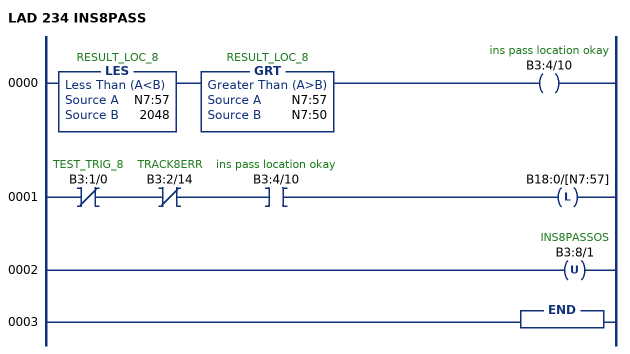
% Rung: 0 %
SOR LES N7:57 2048 GRT N7:57 N7:50 OTE B3:4/10 EOR
%   N7:57  RESULT_LOC_8 %
%   N7:50  INS_8_TRIG_LOC %
%   B3:4/10  "ins pass location okay" %
% Rung: 1 %
SOR XIO B3:1/0 XIO B3:2/14 XIC B3:4/10 OTL B18:0/[N7:57] EOR
%   B3:1/0  TEST_TRIG_8 %
%   B3:2/14  TRACK8ERR %
%   B3:4/10  "ins pass location okay" %
%   B18:0  GOOD2 %
%   N7:57  RESULT_LOC_8 %
% Rung: 2 %
SOR OTU B3:8/1 EOR
%   B3:8/1  INS8PASSOS %
% Rung: 3 %
SOR END EOR

LADDER 235 "INS8FAIL"
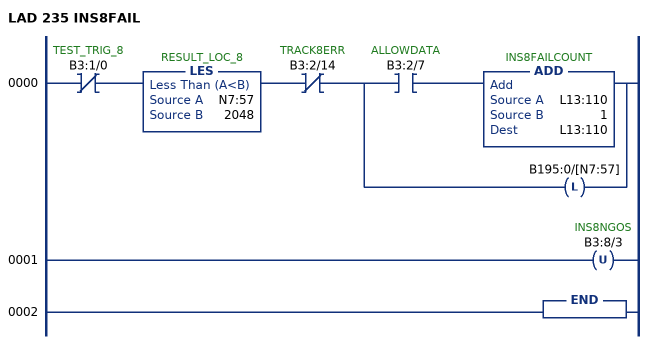
% Rung: 0 %
SOR XIO B3:1/0 LES N7:57 2048 XIO B3:2/14 BST XIC B3:2/7 ADD L13:110 1 L13:110 NXB OTL B195:0/[N7:57] BND EOR
%   B3:1/0  TEST_TRIG_8 %
%   N7:57  RESULT_LOC_8 %
%   B3:2/14  TRACK8ERR %
%   B3:2/7  ALLOWDATA %
%   L13:110  INS8FAILCOUNT %
%   B195:0  TOP_NG %
% Rung: 1 %
SOR OTU B3:8/3 EOR
%   B3:8/3  INS8NGOS %
% Rung: 2 %
SOR END EOR

LADDER 236 "INS8ACQ"
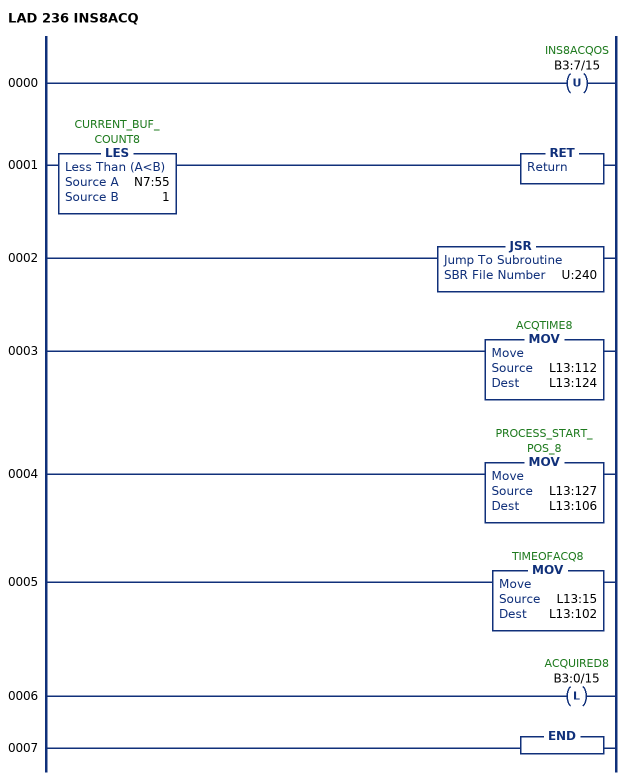
% Rung: 0 %
SOR OTU B3:7/15 EOR
%   B3:7/15  INS8ACQOS %
% Rung: 1 %
SOR LES N7:55 1 RET EOR
%   N7:55  CURRENT_BUF_COUNT8 %
% Rung: 2 %
SOR JSR U:240 EOR
% Rung: 3 %
SOR MOV L13:112 L13:124 EOR
%   L13:112  TIME_SPAN8 %
%   L13:124  ACQTIME8 %
% Rung: 4 %
SOR MOV L13:127 L13:106 EOR
%   L13:127  PULLED_POSITION8 %
%   L13:106  PROCESS_START_POS_8 %
% Rung: 5 %
SOR MOV L13:15 L13:102 EOR
%   L13:15  TOP_TIME %
%   L13:102  TIMEOFACQ8 %
% Rung: 6 %
SOR OTL B3:0/15 EOR
%   B3:0/15  ACQUIRED8 %
% Rung: 7 %
SOR END EOR

LADDER 237 "Q8TIMETEST"
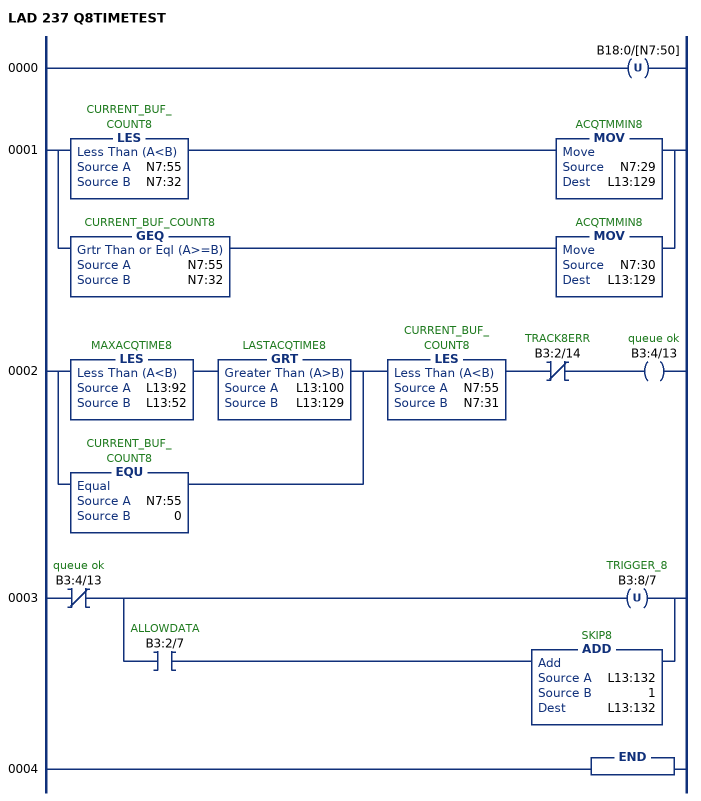
% Rung: 0 %
SOR OTU B18:0/[N7:50] EOR
%   B18:0  GOOD2 %
%   N7:50  INS_8_TRIG_LOC %
% Rung: 1 %
SOR BST LES N7:55 N7:32 MOV N7:29 L13:129 NXB GEQ N7:55 N7:32 MOV N7:30 L13:129 BND EOR
%   N7:55  CURRENT_BUF_COUNT8 %
%   N7:32  BUF_CAM_LIMIT %
%   N7:29  CAM_BUF_ACQ_TM %
%   L13:129  ACQTMMIN8 %
%   N7:30  PC_BUF_ACQ_TM %
% Rung: 2 %
SOR BST LES L13:92 L13:52 GRT L13:100 L13:129 NXB EQU N7:55 0 BND LES N7:55 N7:31 XIO B3:2/14 OTE B3:4/13 EOR
%   L13:92  MAXACQTIME8 %
%   L13:52  ACQTIMELIMIT %
%   L13:100  LASTACQTIME8 %
%   L13:129  ACQTMMIN8 %
%   N7:55  CURRENT_BUF_COUNT8 %
%   N7:31  MAX_BUFF_CT  "maximum buffers" %
%   B3:2/14  TRACK8ERR %
%   B3:4/13  "queue ok" %
% Rung: 3 %
SOR XIO B3:4/13 BST OTU B3:8/7 NXB XIC B3:2/7 ADD L13:132 1 L13:132 BND EOR
%   B3:4/13  "queue ok" %
%   B3:8/7  TRIGGER_8 %
%   B3:2/7  ALLOWDATA %
%   L13:132  SKIP8 %
% Rung: 4 %
SOR END EOR

LADDER 238 "INS8TRIG"
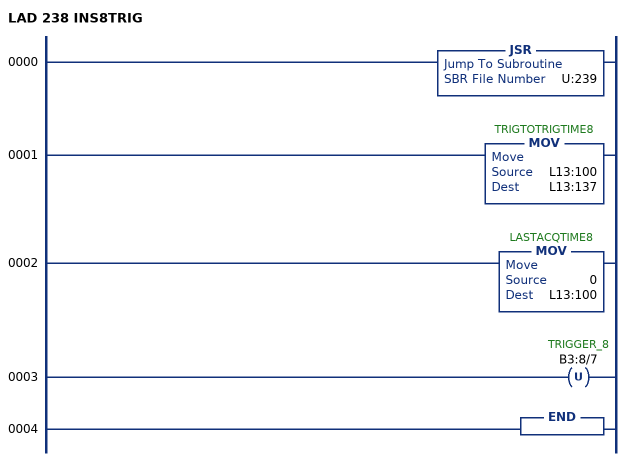
% Rung: 0 %
SOR JSR U:239 EOR
% Rung: 1 %
SOR MOV L13:100 L13:137 EOR
%   L13:100  LASTACQTIME8 %
%   L13:137  TRIGTOTRIGTIME8 %
% Rung: 2 %
SOR MOV 0 L13:100 EOR
%   L13:100  LASTACQTIME8 %
% Rung: 3 %
SOR OTU B3:8/7 EOR
%   B3:8/7  TRIGGER_8 %
% Rung: 4 %
SOR END EOR

LADDER 239 "FIFO8SET"
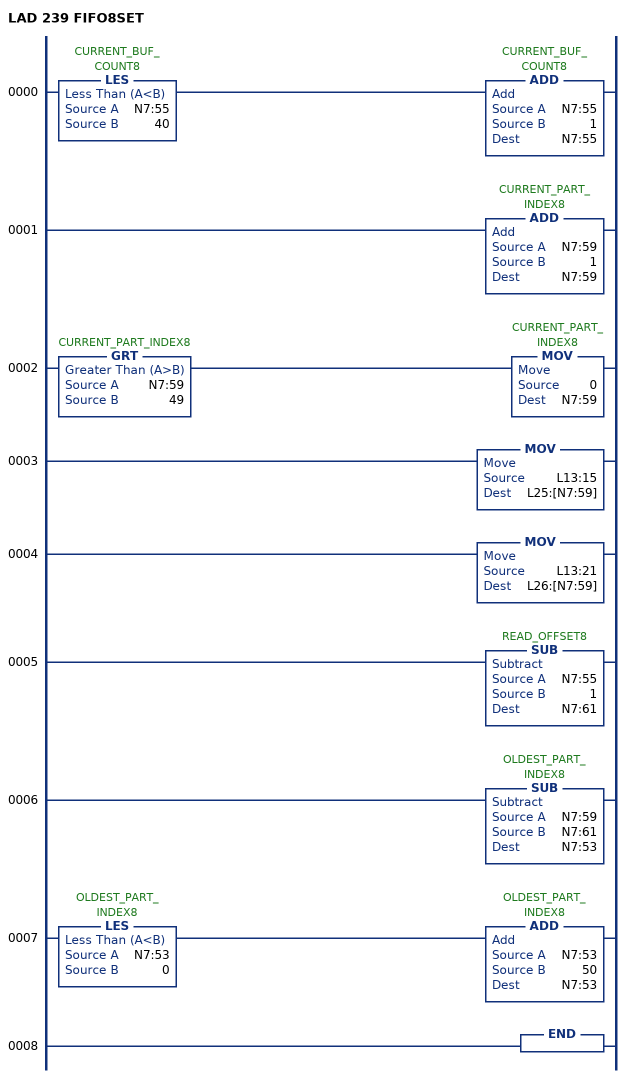
% Rung: 0 %
SOR LES N7:55 40 ADD N7:55 1 N7:55 EOR
%   N7:55  CURRENT_BUF_COUNT8 %
% Rung: 1 %
SOR ADD N7:59 1 N7:59 EOR
%   N7:59  CURRENT_PART_INDEX8 %
% Rung: 2 %
SOR GRT N7:59 49 MOV 0 N7:59 EOR
%   N7:59  CURRENT_PART_INDEX8 %
% Rung: 3 %
SOR MOV L13:15 L25:[N7:59] EOR
%   L13:15  TOP_TIME %
%   N7:59  CURRENT_PART_INDEX8 %
% Rung: 4 %
SOR MOV L13:21 L26:[N7:59] EOR
%   L13:21  TOP_POSITION %
%   N7:59  CURRENT_PART_INDEX8 %
% Rung: 5 %
SOR SUB N7:55 1 N7:61 EOR
%   N7:55  CURRENT_BUF_COUNT8 %
%   N7:61  READ_OFFSET8 %
% Rung: 6 %
SOR SUB N7:59 N7:61 N7:53 EOR
%   N7:59  CURRENT_PART_INDEX8 %
%   N7:61  READ_OFFSET8 %
%   N7:53  OLDEST_PART_INDEX8 %
% Rung: 7 %
SOR LES N7:53 0 ADD N7:53 50 N7:53 EOR
%   N7:53  OLDEST_PART_INDEX8 %
% Rung: 8 %
SOR END EOR

LADDER 240 "FIFO8GET"
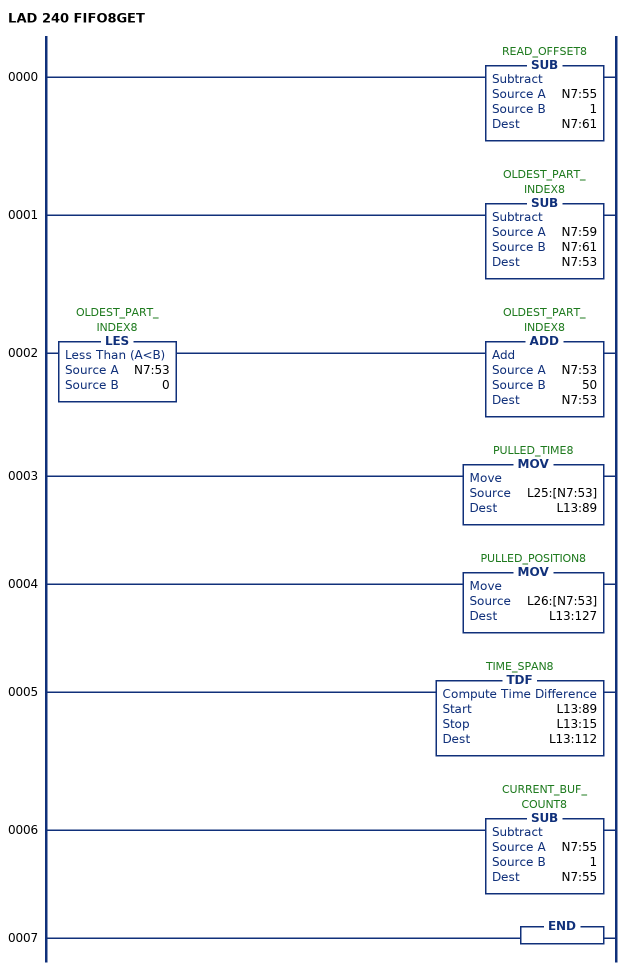
% Rung: 0 %
SOR SUB N7:55 1 N7:61 EOR
%   N7:55  CURRENT_BUF_COUNT8 %
%   N7:61  READ_OFFSET8 %
% Rung: 1 %
SOR SUB N7:59 N7:61 N7:53 EOR
%   N7:59  CURRENT_PART_INDEX8 %
%   N7:61  READ_OFFSET8 %
%   N7:53  OLDEST_PART_INDEX8 %
% Rung: 2 %
SOR LES N7:53 0 ADD N7:53 50 N7:53 EOR
%   N7:53  OLDEST_PART_INDEX8 %
% Rung: 3 %
SOR MOV L25:[N7:53] L13:89 EOR
%   N7:53  OLDEST_PART_INDEX8 %
%   L13:89  PULLED_TIME8 %
% Rung: 4 %
SOR MOV L26:[N7:53] L13:127 EOR
%   N7:53  OLDEST_PART_INDEX8 %
%   L13:127  PULLED_POSITION8 %
% Rung: 5 %
SOR TDF L13:89 L13:15 L13:112 EOR
%   L13:89  PULLED_TIME8 %
%   L13:15  TOP_TIME %
%   L13:112  TIME_SPAN8 %
% Rung: 6 %
SOR SUB N7:55 1 N7:55 EOR
%   N7:55  CURRENT_BUF_COUNT8 %
% Rung: 7 %
SOR END EOR

LADDER 241 "INSDATA8"
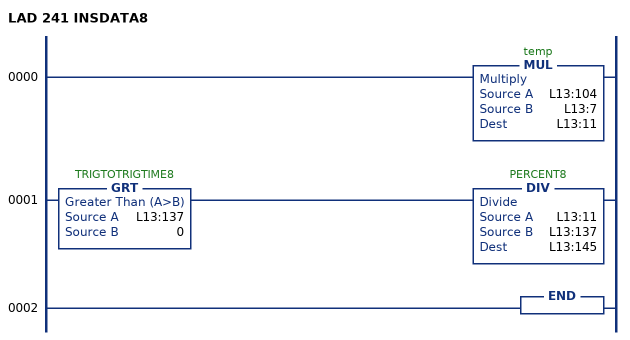
% Rung: 0 %
SOR MUL L13:104 L13:7 L13:11 EOR
%   L13:104  PROCESSTIME8 %
%   L13:7  PERCENT_MULTIPLYER %
%   L13:11  "temp" %
% Rung: 1 %
SOR GRT L13:137 0 DIV L13:11 L13:137 L13:145 EOR
%   L13:137  TRIGTOTRIGTIME8 %
%   L13:11  "temp" %
%   L13:145  PERCENT8 %
% Rung: 2 %
SOR END EOR

LADDER 242 "TESTFAULT8"
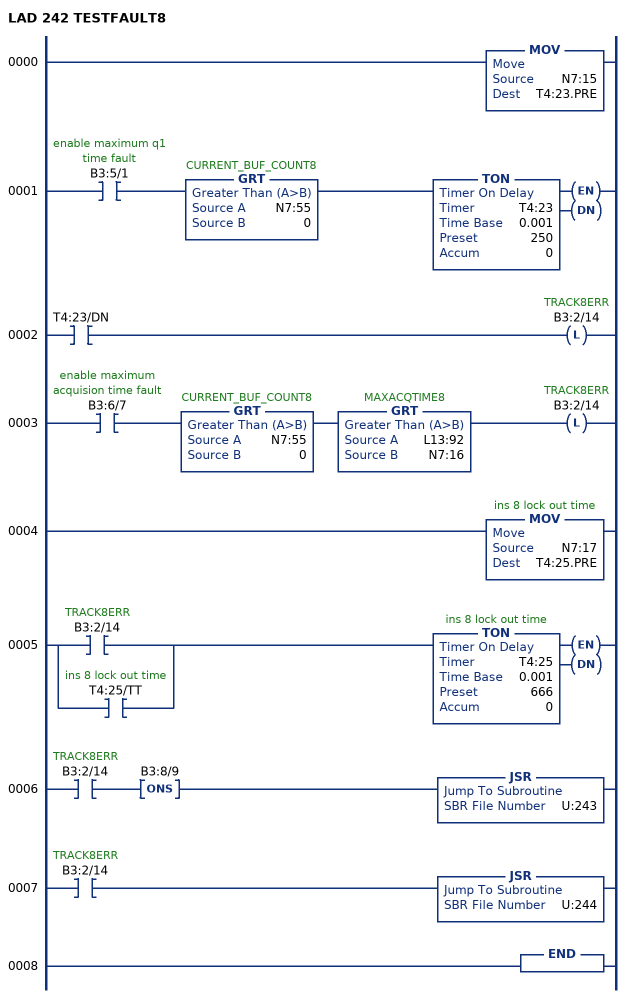
% Rung: 0 %
SOR MOV N7:15 T4:23.PRE EOR
%   N7:15  "max allowed ms time for q to be above 1 if safe fault is used" %
% Rung: 1 %
SOR XIC B3:5/1 GRT N7:55 0 TON T4:23 0.001 250 0 EOR
%   B3:5/1  "enable maximum q1 time fault" %
%   N7:55  CURRENT_BUF_COUNT8 %
% Rung: 2 %
SOR XIC T4:23/DN OTL B3:2/14 EOR
%   B3:2/14  TRACK8ERR %
% Rung: 3 %
SOR XIC B3:6/7 GRT N7:55 0 GRT L13:92 N7:16 OTL B3:2/14 EOR
%   B3:6/7  "enable maximum acquision time fault" %
%   N7:55  CURRENT_BUF_COUNT8 %
%   L13:92  MAXACQTIME8 %
%   N7:16  ACQUIRE_TIME_LIMIT  "maximum of the longest acquire time allowed if maximum acquire time fault is enabled" %
%   B3:2/14  TRACK8ERR %
% Rung: 4 %
SOR MOV N7:17 T4:25.PRE EOR
%   N7:17  "ms time setting to lock out inspection to give all pending images a chance to clear" %
%   T4:25  "ins 8 lock out time" %
% Rung: 5 %
SOR BST XIC B3:2/14 NXB XIC T4:25/TT BND TON T4:25 0.001 666 0 EOR
%   B3:2/14  TRACK8ERR %
%   T4:25  "ins 8 lock out time" %
% Rung: 6 %
SOR XIC B3:2/14 ONS B3:8/9 JSR U:243 EOR
%   B3:2/14  TRACK8ERR %
% Rung: 7 %
SOR XIC B3:2/14 JSR U:244 EOR
%   B3:2/14  TRACK8ERR %
% Rung: 8 %
SOR END EOR

LADDER 243 "INS8FIX1"
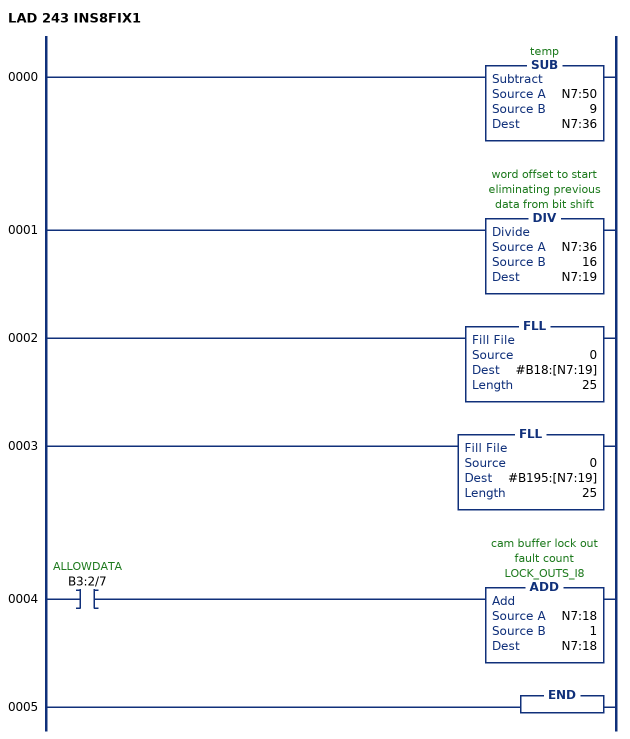
% Rung: 0 %
SOR SUB N7:50 9 N7:36 EOR
%   N7:50  INS_8_TRIG_LOC %
%   N7:36  "temp" %
% Rung: 1 %
SOR DIV N7:36 16 N7:19 EOR
%   N7:36  "temp" %
%   N7:19  "word offset to start eliminating previous data from bit shift" %
% Rung: 2 %
SOR FLL 0 #B18:[N7:19] 25 EOR
%   N7:19  "word offset to start eliminating previous data from bit shift" %
% Rung: 3 %
SOR FLL 0 #B195:[N7:19] 25 EOR
%   N7:19  "word offset to start eliminating previous data from bit shift" %
% Rung: 4 %
SOR XIC B3:2/7 ADD N7:18 1 N7:18 EOR
%   B3:2/7  ALLOWDATA %
%   N7:18  LOCK_OUTS_I8  "cam buffer lock out fault count" %
% Rung: 5 %
SOR END EOR

LADDER 244 "INS8FIX2"
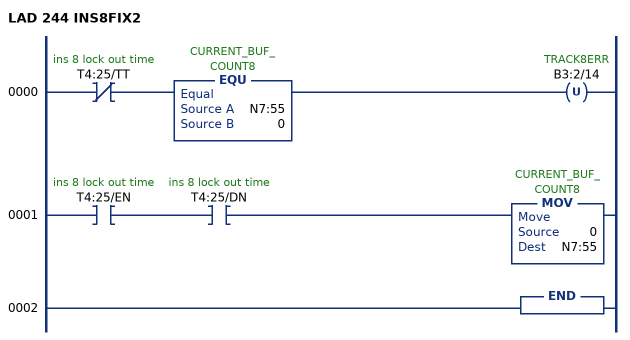
% Rung: 0 %
SOR XIO T4:25/TT EQU N7:55 0 OTU B3:2/14 EOR
%   T4:25  "ins 8 lock out time" %
%   N7:55  CURRENT_BUF_COUNT8 %
%   B3:2/14  TRACK8ERR %
% Rung: 1 %
SOR XIC T4:25/EN XIC T4:25/DN MOV 0 N7:55 EOR
%   T4:25  "ins 8 lock out time" %
%   N7:55  CURRENT_BUF_COUNT8 %
% Rung: 2 %
SOR END EOR

LADDER 249 "PASS BLOW"
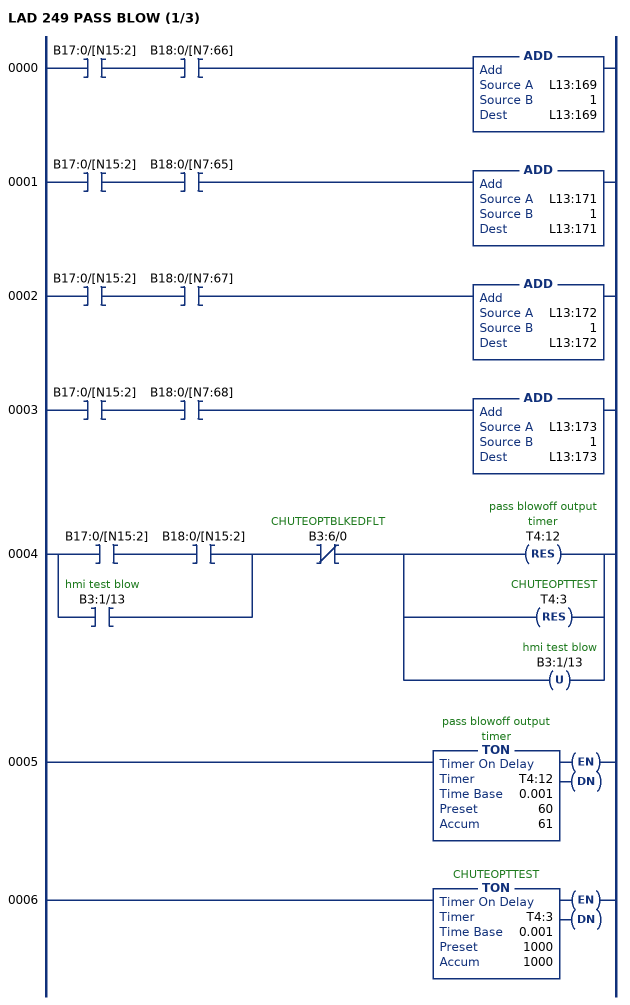
% Rung: 0 %
SOR XIC B17:0/[N15:2] XIC B18:0/[N7:66] ADD L13:169 1 L13:169 EOR
%   B17:0  GOOD1 %
%   N15:2  BLOW_PT %
%   B18:0  GOOD2 %
%   N7:66  P2 %
% Rung: 1 %
SOR XIC B17:0/[N15:2] XIC B18:0/[N7:65] ADD L13:171 1 L13:171 EOR
%   B17:0  GOOD1 %
%   N15:2  BLOW_PT %
%   B18:0  GOOD2 %
%   N7:65  P1 %
% Rung: 2 %
SOR XIC B17:0/[N15:2] XIC B18:0/[N7:67] ADD L13:172 1 L13:172 EOR
%   B17:0  GOOD1 %
%   N15:2  BLOW_PT %
%   B18:0  GOOD2 %
%   N7:67  M1 %
% Rung: 3 %
SOR XIC B17:0/[N15:2] XIC B18:0/[N7:68] ADD L13:173 1 L13:173 EOR
%   B17:0  GOOD1 %
%   N15:2  BLOW_PT %
%   B18:0  GOOD2 %
%   N7:68  M2 %
% Rung: 4 %
SOR BST XIC B17:0/[N15:2] XIC B18:0/[N15:2] NXB XIC B3:1/13 BND XIO B3:6/0 BST RES T4:12 NXB RES T4:3 NXB OTU B3:1/13 BND EOR
%   B17:0  GOOD1 %
%   N15:2  BLOW_PT %
%   B18:0  GOOD2 %
%   B3:1/13  "hmi test blow" %
%   B3:6/0  CHUTEOPTBLKEDFLT %
%   T4:12  "pass blowoff output timer" %
%   T4:3  CHUTEOPTTEST %
% Rung: 5 %
SOR TON T4:12 0.001 60 61 EOR
%   T4:12  "pass blowoff output timer" %
% Rung: 6 %
SOR TON T4:3 0.001 1000 1000 EOR
%   T4:3  CHUTEOPTTEST %

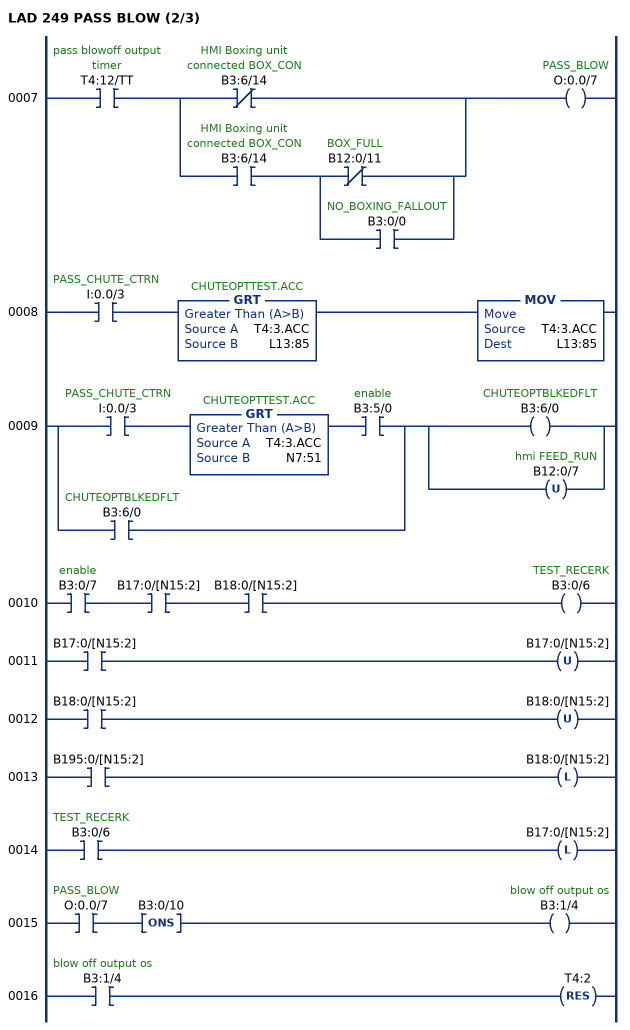
% Rung: 7 %
SOR XIC T4:12/TT BST XIO B3:6/14 NXB XIC B3:6/14 BST XIO B12:0/11 NXB XIC B3:0/0 BND BND OTE O:0.0/7 EOR
%   T4:12  "pass blowoff output timer" %
%   B3:6/14  BOX_CON  "HMI Boxing unit connected" %
%   B12:0/11  BOX_FULL %
%   B3:0/0  NO_BOXING_FALLOUT %
%   O:0.0/7  PASS_BLOW %
% Rung: 8 %
SOR XIC I:0.0/3 GRT T4:3.ACC L13:85 MOV T4:3.ACC L13:85 EOR
%   I:0.0/3  PASS_CHUTE_CTRN %
%   T4:3  CHUTEOPTTEST %
% Rung: 9 %
SOR BST XIC I:0.0/3 GRT T4:3.ACC N7:51 XIC B3:5/0 NXB XIC B3:6/0 BND BST OTE B3:6/0 NXB OTU B12:0/7 BND EOR
%   I:0.0/3  PASS_CHUTE_CTRN %
%   T4:3  CHUTEOPTTEST %
%   B3:5/0  "enable" %
%   B3:6/0  CHUTEOPTBLKEDFLT %
%   B12:0/7  FEED_RUN  "hmi" %
% Rung: 10 %
SOR XIC B3:0/7 XIC B17:0/[N15:2] XIC B18:0/[N15:2] OTE B3:0/6 EOR
%   B3:0/7  "enable" %
%   B17:0  GOOD1 %
%   N15:2  BLOW_PT %
%   B18:0  GOOD2 %
%   B3:0/6  TEST_RECERK %
% Rung: 11 %
SOR XIC B17:0/[N15:2] OTU B17:0/[N15:2] EOR
%   B17:0  GOOD1 %
%   N15:2  BLOW_PT %
% Rung: 12 %
SOR XIC B18:0/[N15:2] OTU B18:0/[N15:2] EOR
%   B18:0  GOOD2 %
%   N15:2  BLOW_PT %
% Rung: 13 %
SOR XIC B195:0/[N15:2] OTL B18:0/[N15:2] EOR
%   B195:0  TOP_NG %
%   N15:2  BLOW_PT %
%   B18:0  GOOD2 %
% Rung: 14 %
SOR XIC B3:0/6 OTL B17:0/[N15:2] EOR
%   B3:0/6  TEST_RECERK %
%   B17:0  GOOD1 %
%   N15:2  BLOW_PT %
% Rung: 15 %
SOR XIC O:0.0/7 ONS B3:0/10 OTE B3:1/4 EOR
%   O:0.0/7  PASS_BLOW %
%   B3:1/4  "blow off output os" %
% Rung: 16 %
SOR XIC B3:1/4 RES T4:2 EOR
%   B3:1/4  "blow off output os" %

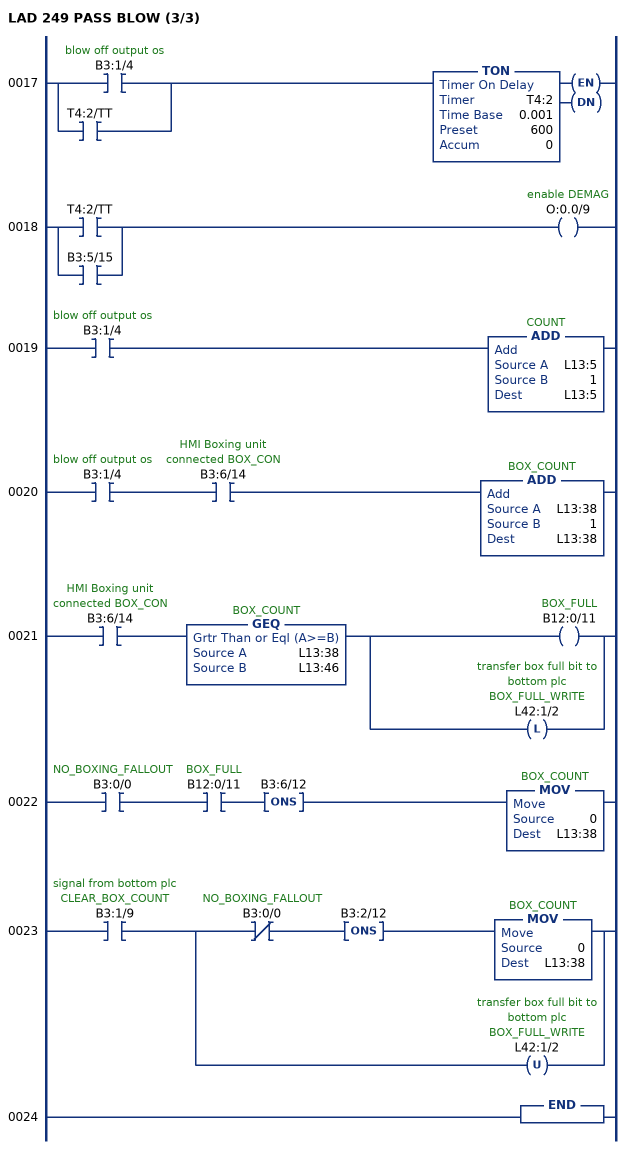
% Rung: 17 %
SOR BST XIC B3:1/4 NXB XIC T4:2/TT BND TON T4:2 0.001 600 0 EOR
%   B3:1/4  "blow off output os" %
% Rung: 18 %
SOR BST XIC T4:2/TT NXB XIC B3:5/15 BND OTE O:0.0/9 EOR
%   O:0.0/9  DEMAG  "enable" %
% Rung: 19 %
SOR XIC B3:1/4 ADD L13:5 1 L13:5 EOR
%   B3:1/4  "blow off output os" %
%   L13:5  COUNT %
% Rung: 20 %
SOR XIC B3:1/4 XIC B3:6/14 ADD L13:38 1 L13:38 EOR
%   B3:1/4  "blow off output os" %
%   B3:6/14  BOX_CON  "HMI Boxing unit connected" %
%   L13:38  BOX_COUNT %
% Rung: 21 %
SOR XIC B3:6/14 GEQ L13:38 L13:46 BST OTE B12:0/11 NXB OTL L42:1/2 BND EOR
%   B3:6/14  BOX_CON  "HMI Boxing unit connected" %
%   L13:38  BOX_COUNT %
%   L13:46  BOX_LIMIT  "box count setpoint" %
%   B12:0/11  BOX_FULL %
%   L42:1/2  BOX_FULL_WRITE  "transfer box full bit to bottom plc" %
% Rung: 22 %
SOR XIC B3:0/0 XIC B12:0/11 ONS B3:6/12 MOV 0 L13:38 EOR
%   B3:0/0  NO_BOXING_FALLOUT %
%   B12:0/11  BOX_FULL %
%   L13:38  BOX_COUNT %
% Rung: 23 %
SOR XIC B3:1/9 BST XIO B3:0/0 ONS B3:2/12 MOV 0 L13:38 NXB OTU L42:1/2 BND EOR
%   B3:1/9  CLEAR_BOX_COUNT  "signal from bottom plc" %
%   B3:0/0  NO_BOXING_FALLOUT %
%   L13:38  BOX_COUNT %
%   L42:1/2  BOX_FULL_WRITE  "transfer box full bit to bottom plc" %
% Rung: 24 %
SOR END EOR

LADDER 250 "RECERK"
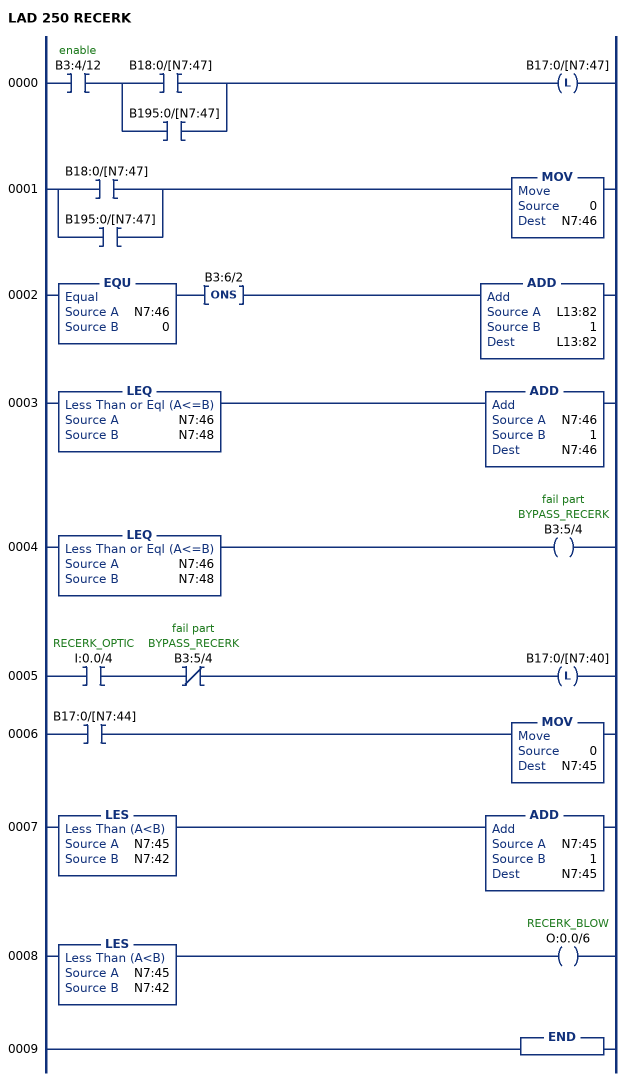
% Rung: 0 %
SOR XIC B3:4/12 BST XIC B18:0/[N7:47] NXB XIC B195:0/[N7:47] BND OTL B17:0/[N7:47] EOR
%   B3:4/12  "enable" %
%   B18:0  GOOD2 %
%   N7:47  RECERK_BLOCKOPTIC_PT %
%   B195:0  TOP_NG %
%   B17:0  GOOD1 %
% Rung: 1 %
SOR BST XIC B18:0/[N7:47] NXB XIC B195:0/[N7:47] BND MOV 0 N7:46 EOR
%   B18:0  GOOD2 %
%   N7:47  RECERK_BLOCKOPTIC_PT %
%   B195:0  TOP_NG %
% Rung: 2 %
SOR EQU N7:46 0 ONS B3:6/2 ADD L13:82 1 L13:82 EOR
% Rung: 3 %
SOR LEQ N7:46 N7:48 ADD N7:46 1 N7:46 EOR
%   N7:48  RECERK_BLK_BLOW_DIST %
% Rung: 4 %
SOR LEQ N7:46 N7:48 OTE B3:5/4 EOR
%   N7:48  RECERK_BLK_BLOW_DIST %
%   B3:5/4  BYPASS_RECERK  "fail part" %
% Rung: 5 %
SOR XIC I:0.0/4 XIO B3:5/4 OTL B17:0/[N7:40] EOR
%   I:0.0/4  RECERK_OPTIC %
%   B3:5/4  BYPASS_RECERK  "fail part" %
%   B17:0  GOOD1 %
%   N7:40  RECERK_OPTIC_POS %
% Rung: 6 %
SOR XIC B17:0/[N7:44] MOV 0 N7:45 EOR
%   B17:0  GOOD1 %
%   N7:44  RECERK_BLOW_POS  "adjusted for blow length" %
% Rung: 7 %
SOR LES N7:45 N7:42 ADD N7:45 1 N7:45 EOR
%   N7:42  RECERK_BLOW_LENGTH %
% Rung: 8 %
SOR LES N7:45 N7:42 OTE O:0.0/6 EOR
%   N7:42  RECERK_BLOW_LENGTH %
%   O:0.0/6  RECERK_BLOW %
% Rung: 9 %
SOR END EOR

LADDER 251 "RECERK SET"
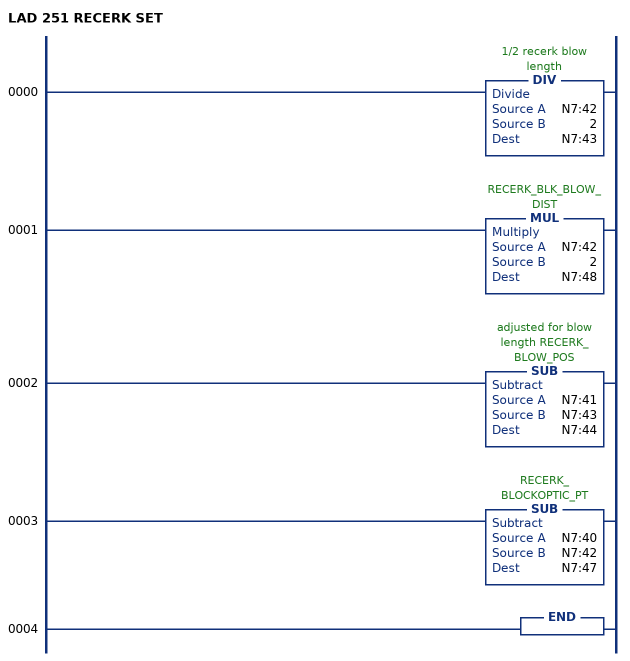
% Rung: 0 %
SOR DIV N7:42 2 N7:43 EOR
%   N7:42  RECERK_BLOW_LENGTH %
%   N7:43  "1/2 recerk blow length" %
% Rung: 1 %
SOR MUL N7:42 2 N7:48 EOR
%   N7:42  RECERK_BLOW_LENGTH %
%   N7:48  RECERK_BLK_BLOW_DIST %
% Rung: 2 %
SOR SUB N7:41 N7:43 N7:44 EOR
%   N7:41  RECERK_BLOW_POS_HMI  "recerk blow position set from hmi" %
%   N7:43  "1/2 recerk blow length" %
%   N7:44  RECERK_BLOW_POS  "adjusted for blow length" %
% Rung: 3 %
SOR SUB N7:40 N7:42 N7:47 EOR
%   N7:40  RECERK_OPTIC_POS %
%   N7:42  RECERK_BLOW_LENGTH %
%   N7:47  RECERK_BLOCKOPTIC_PT %
% Rung: 4 %
SOR END EOR

LADDER 252 "RATE1"
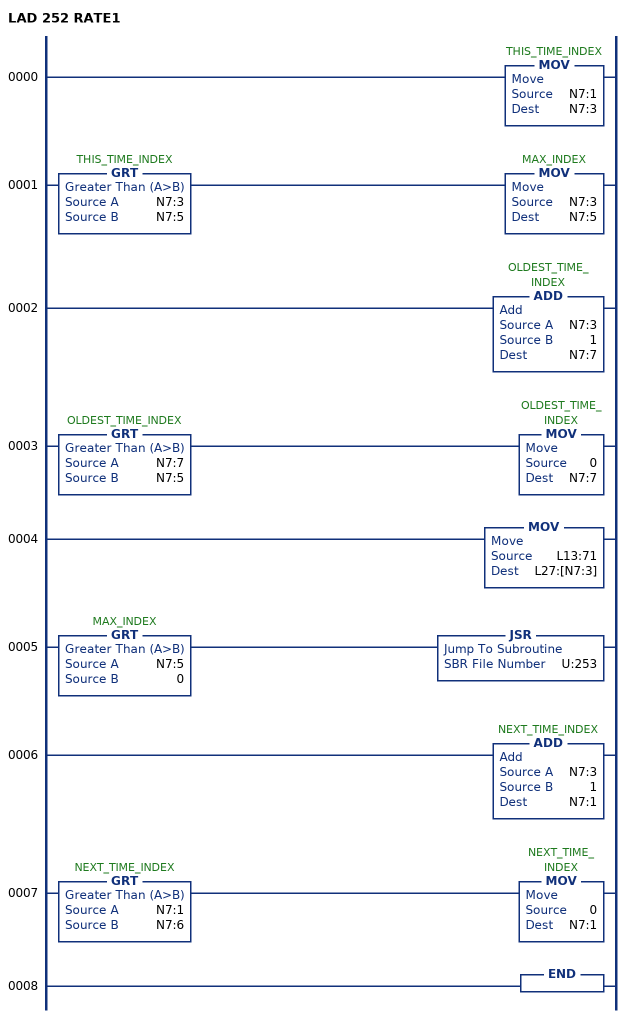
% Rung: 0 %
SOR MOV N7:1 N7:3 EOR
%   N7:1  NEXT_TIME_INDEX %
%   N7:3  THIS_TIME_INDEX %
% Rung: 1 %
SOR GRT N7:3 N7:5 MOV N7:3 N7:5 EOR
%   N7:3  THIS_TIME_INDEX %
%   N7:5  MAX_INDEX %
% Rung: 2 %
SOR ADD N7:3 1 N7:7 EOR
%   N7:3  THIS_TIME_INDEX %
%   N7:7  OLDEST_TIME_INDEX %
% Rung: 3 %
SOR GRT N7:7 N7:5 MOV 0 N7:7 EOR
%   N7:7  OLDEST_TIME_INDEX %
%   N7:5  MAX_INDEX %
% Rung: 4 %
SOR MOV L13:71 L27:[N7:3] EOR
%   L13:71  HSC_TIME %
%   N7:3  THIS_TIME_INDEX %
% Rung: 5 %
SOR GRT N7:5 0 JSR U:253 EOR
%   N7:5  MAX_INDEX %
% Rung: 6 %
SOR ADD N7:3 1 N7:1 EOR
%   N7:3  THIS_TIME_INDEX %
%   N7:1  NEXT_TIME_INDEX %
% Rung: 7 %
SOR GRT N7:1 N7:6 MOV 0 N7:1 EOR
%   N7:1  NEXT_TIME_INDEX %
%   N7:6  UPPER_INDEX_LIMIT  "buffer count 1" %
% Rung: 8 %
SOR END EOR

LADDER 253 "RATE2"
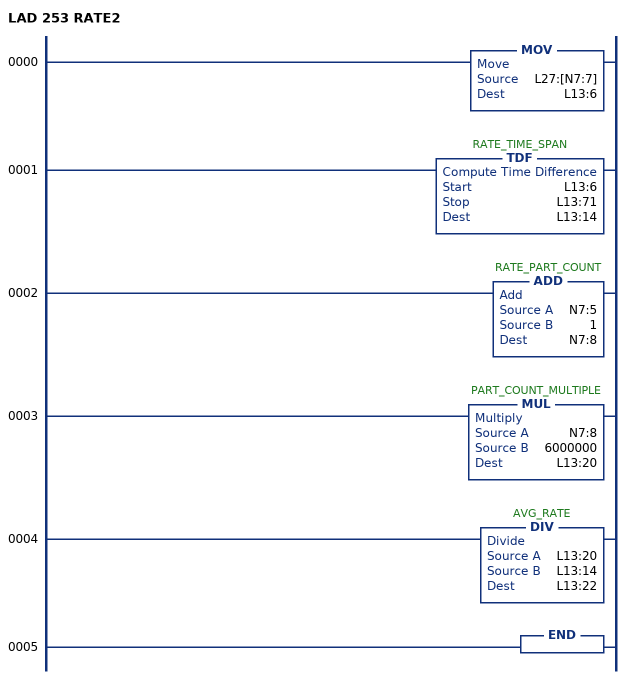
% Rung: 0 %
SOR MOV L27:[N7:7] L13:6 EOR
%   N7:7  OLDEST_TIME_INDEX %
% Rung: 1 %
SOR TDF L13:6 L13:71 L13:14 EOR
%   L13:71  HSC_TIME %
%   L13:14  RATE_TIME_SPAN %
% Rung: 2 %
SOR ADD N7:5 1 N7:8 EOR
%   N7:5  MAX_INDEX %
%   N7:8  RATE_PART_COUNT %
% Rung: 3 %
SOR MUL N7:8 6000000 L13:20 EOR
%   N7:8  RATE_PART_COUNT %
%   L13:20  PART_COUNT_MULTIPLE %
% Rung: 4 %
SOR DIV L13:20 L13:14 L13:22 EOR
%   L13:20  PART_COUNT_MULTIPLE %
%   L13:14  RATE_TIME_SPAN %
%   L13:22  AVG_RATE %
% Rung: 5 %
SOR END EOR

LADDER 254 "RESET RATE"
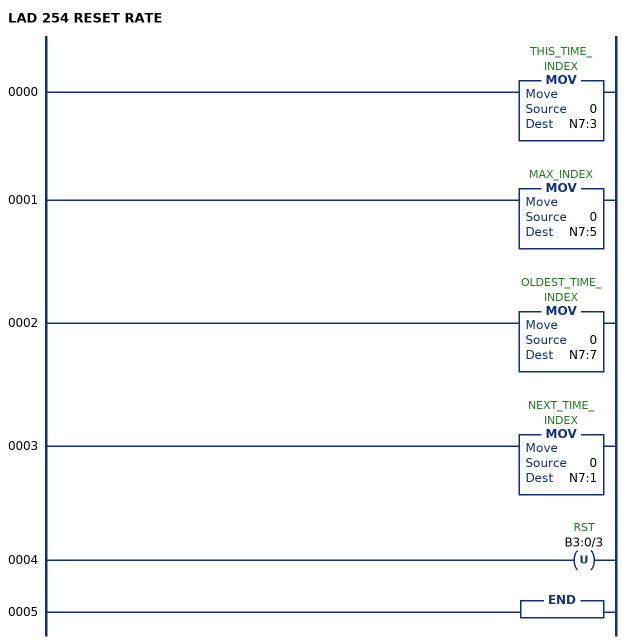
% Rung: 0 %
SOR MOV 0 N7:3 EOR
%   N7:3  THIS_TIME_INDEX %
% Rung: 1 %
SOR MOV 0 N7:5 EOR
%   N7:5  MAX_INDEX %
% Rung: 2 %
SOR MOV 0 N7:7 EOR
%   N7:7  OLDEST_TIME_INDEX %
% Rung: 3 %
SOR MOV 0 N7:1 EOR
%   N7:1  NEXT_TIME_INDEX %
% Rung: 4 %
SOR OTU B3:0/3 EOR
%   B3:0/3  RST %
% Rung: 5 %
SOR END EOR

LADDER 255 "UNUSED"
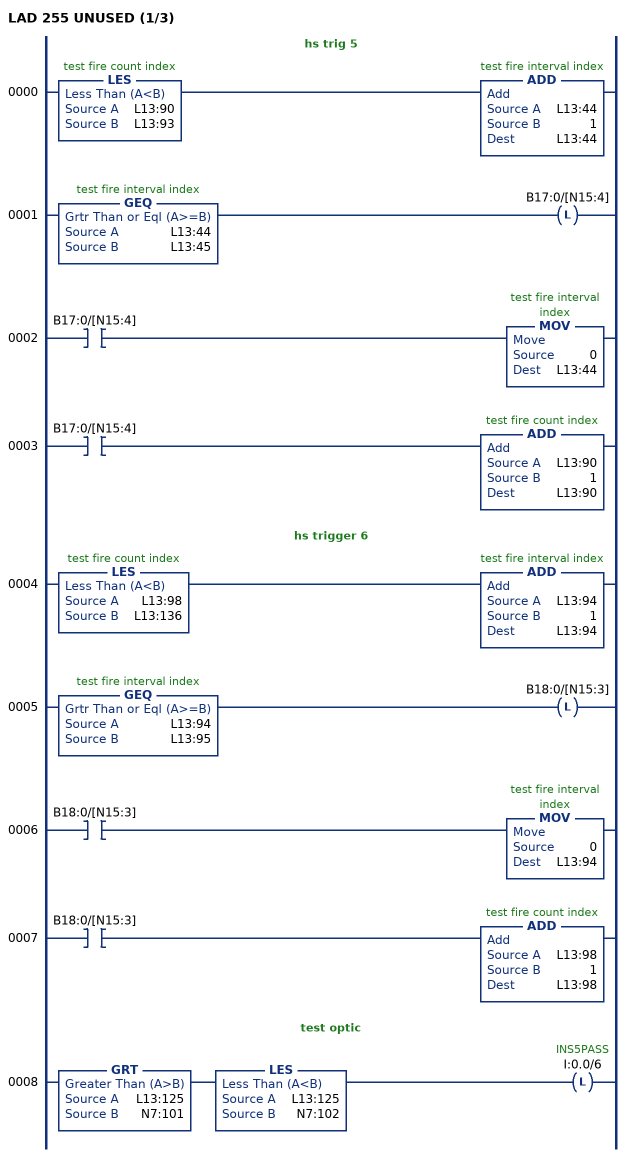
% Rung: 0 %
% TITLE: hs trig 5 %
SOR LES L13:90 L13:93 ADD L13:44 1 L13:44 EOR
%   L13:90  "test fire count index" %
%   L13:93  "test fire count" %
%   L13:44  "test fire interval index" %
% Rung: 1 %
SOR GEQ L13:44 L13:45 OTL B17:0/[N15:4] EOR
%   L13:44  "test fire interval index" %
%   L13:45  "test fire interval" %
%   B17:0  GOOD1 %
%   N15:4  INS_5_TRIG_LOC %
% Rung: 2 %
SOR XIC B17:0/[N15:4] MOV 0 L13:44 EOR
%   B17:0  GOOD1 %
%   N15:4  INS_5_TRIG_LOC %
%   L13:44  "test fire interval index" %
% Rung: 3 %
SOR XIC B17:0/[N15:4] ADD L13:90 1 L13:90 EOR
%   B17:0  GOOD1 %
%   N15:4  INS_5_TRIG_LOC %
%   L13:90  "test fire count index" %
% Rung: 4 %
% TITLE: hs trigger 6 %
SOR LES L13:98 L13:136 ADD L13:94 1 L13:94 EOR
%   L13:98  "test fire count index" %
%   L13:136  "test fire count" %
%   L13:94  "test fire interval index" %
% Rung: 5 %
SOR GEQ L13:94 L13:95 OTL B18:0/[N15:3] EOR
%   L13:94  "test fire interval index" %
%   L13:95  "test fire interval" %
%   B18:0  GOOD2 %
%   N15:3  INS_6_TRIG_LOC %
% Rung: 6 %
SOR XIC B18:0/[N15:3] MOV 0 L13:94 EOR
%   B18:0  GOOD2 %
%   N15:3  INS_6_TRIG_LOC %
%   L13:94  "test fire interval index" %
% Rung: 7 %
SOR XIC B18:0/[N15:3] ADD L13:98 1 L13:98 EOR
%   B18:0  GOOD2 %
%   N15:3  INS_6_TRIG_LOC %
%   L13:98  "test fire count index" %
% Rung: 8 %
% TITLE: test optic %
SOR GRT L13:125 N7:101 LES L13:125 N7:102 OTL I:0.0/6 EOR
%   I:0.0/6  INS5PASS %

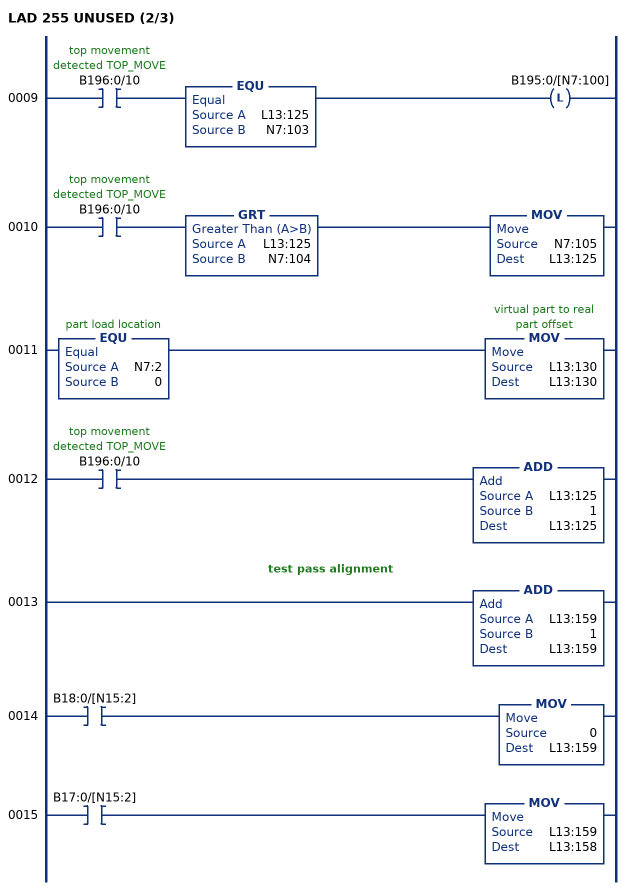
% Rung: 9 %
SOR XIC B196:0/10 EQU L13:125 N7:103 OTL B195:0/[N7:100] EOR
%   B196:0/10  TOP_MOVE  "top movement detected" %
%   B195:0  TOP_NG %
% Rung: 10 %
SOR XIC B196:0/10 GRT L13:125 N7:104 MOV N7:105 L13:125 EOR
%   B196:0/10  TOP_MOVE  "top movement detected" %
% Rung: 11 %
SOR EQU N7:2 0 MOV L13:130 L13:130 EOR
%   N7:2  "part load location" %
%   L13:130  "virtual part to real part offset" %
% Rung: 12 %
SOR XIC B196:0/10 ADD L13:125 1 L13:125 EOR
%   B196:0/10  TOP_MOVE  "top movement detected" %
% Rung: 13 %
% TITLE: test pass alignment %
SOR ADD L13:159 1 L13:159 EOR
% Rung: 14 %
SOR XIC B18:0/[N15:2] MOV 0 L13:159 EOR
%   B18:0  GOOD2 %
%   N15:2  BLOW_PT %
% Rung: 15 %
SOR XIC B17:0/[N15:2] MOV L13:159 L13:158 EOR
%   B17:0  GOOD1 %
%   N15:2  BLOW_PT %

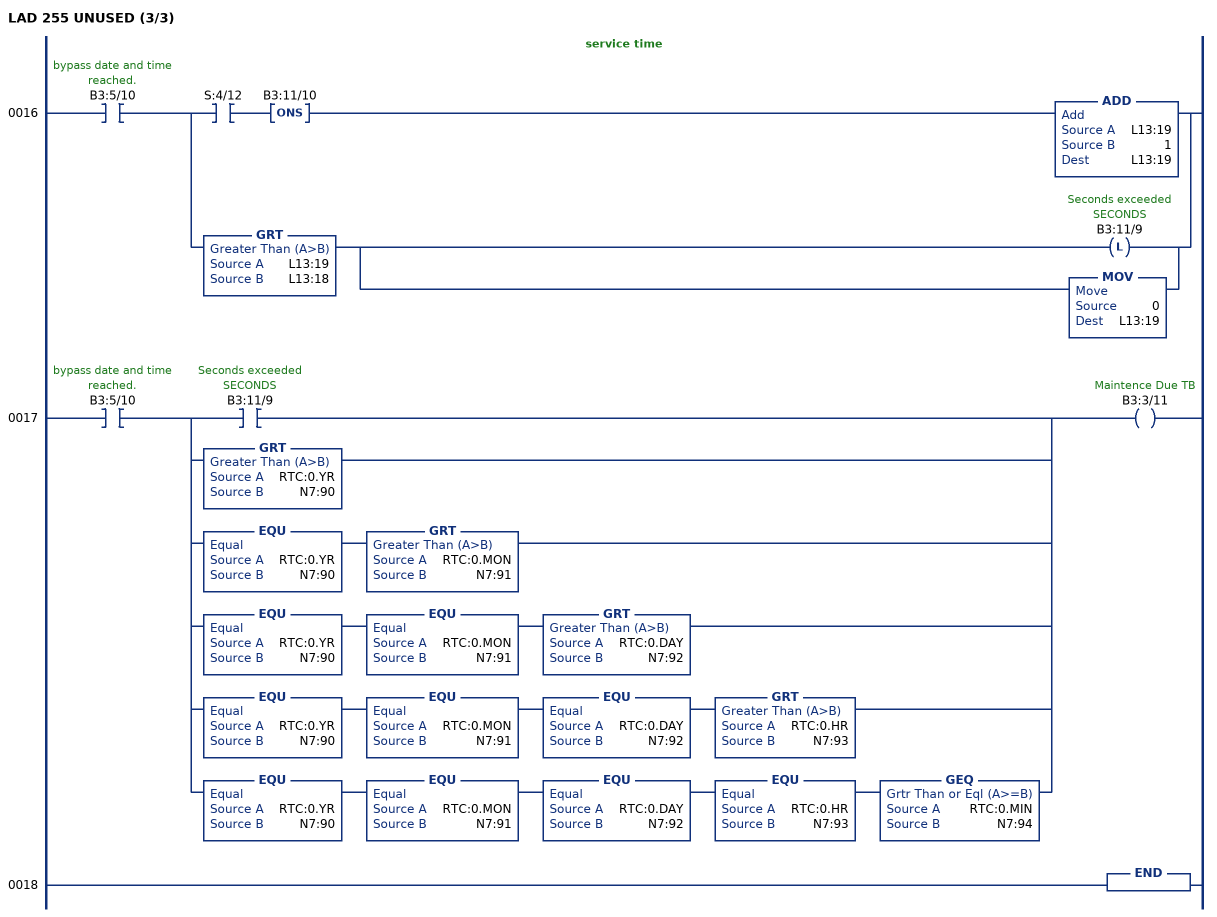
% Rung: 16 %
% TITLE: service time %
SOR XIC B3:5/10 BST XIC S:4/12 ONS B3:11/10 ADD L13:19 1 L13:19 NXB GRT L13:19 L13:18 BST OTL B3:11/9 NXB MOV 0 L13:19 BND BND EOR
%   B3:5/10  "bypass date and time reached." %
%   L13:18  MAX %
%   B3:11/9  SECONDS  "Seconds exceeded" %
% Rung: 17 %
SOR XIC B3:5/10 BST XIC B3:11/9 NXB GRT RTC:0.YR N7:90 NXB EQU RTC:0.YR N7:90 GRT RTC:0.MON N7:91 NXB EQU RTC:0.YR N7:90 EQU RTC:0.MON N7:91 GRT RTC:0.DAY N7:92 NXB EQU RTC:0.YR N7:90 EQU RTC:0.MON N7:91 EQU RTC:0.DAY N7:92 GRT RTC:0.HR N7:93 NXB EQU RTC:0.YR N7:90 EQU RTC:0.MON N7:91 EQU RTC:0.DAY N7:92 EQU RTC:0.HR N7:93 GEQ RTC:0.MIN N7:94 BND OTE B3:3/11 EOR
%   B3:5/10  "bypass date and time reached." %
%   B3:11/9  SECONDS  "Seconds exceeded" %
%   N7:90  RTC %
%   B3:3/11  TB  "Maintence Due" %
% Rung: 18 %
SOR END EOR

OTHER DOCUMENTED ADDRESSES
  B12:0/1  FELL_PARTS_FAULT
  B196:1/2  DOWNTRACK_OPTIC_RUN  "Feed Bowl optic Run Signal after timing delays"
  I:0.0/0  TOP_CONV_ENC_A
  I:0.0/1  TOP_CONV_ENC_B
  I:0.7  "Air Presure Sensor Input Signal"
  L42:0/2  "box full read (unused)"
  L42:1/1  "ps stop write (unused)"
  N15:9  FEED_WHEEL_STOP_TIME
  N197:7  "down track on delay"
  N197:8  "down track off delay"
  O:0.0/0  "spare"
  O:0.0/1  "spare"
  O:0.0/10  "spare"
  O:0.0/11  "spare"
  PFILE:6  "check for part jams"
  PFILE:10  "Bottom belt HSC"
  PFILE:12  "Top belt HSC"
  Q2:55  END_OF_MAIN
  T4:6  FEED_WHEEL_OFF_TIMER  "Delay to shut off feed wheel"
  U:6  "feed"
  U:217  "test trigger"

COMMENTS NOT ATTACHED TO A CURRENT RUNG
  N17:8: ****************************************************************************************************************
    I can not find anywhere in the program where the "Test Spacing From Pickup to Trigger is activated indicating to me that this entire function must not be doing anything in this program at this time.
    ****************************************************************************************************************
  T20:2: The timer used to verify that the part that triggered the top laser optic has passed the bottom camer. needs to be count
  T20:2.ACC: This rung is starting a timer that should be activated directly before the laser optic part presense sensor on the top conveyer and should cause the top optic to be ignored if the bottom camera system didn't pass. however other arrangements must be made if the bottom camera isn't going to be used as is the case with a nut inspection.
  B22:0/0: ***********************
     Bottom Part Syncronizing Logic
    ***********************
    
    This is the point at the bottom of the top conveyor where the part jumps from the bottom conveyor.  This system will then track the part through the top system to the point of the laser optic in order to verify that the part in question has passed the bottom inspection.  I believe that we NEED to include FAILING inspections to eliminate the possibility of a out of position part from passing. LW 072010
  C5:4: tempory counting to verify pass part count with boxing part count.
  B23:0/0: Yet another bit shift load with data in the part position indicating that there was a bottom system part pass as well as a top system part present at this location.
    
    verified works w/bypassed 071910 and unbypassed 072010
  I:0.0/8: special rung for testing. This rung can simulate a pass signal. It will not be timed correctly.
  F8:13: *************************
    Loads Side Camera Passing data into a bit shift
    *************************
    
    loads passing data bit into passing data bit shift register at the part present cl.
  B3:7/9: ************************************
     The next 3 rungs appear to do nothing
    ***********************************
  B11:0/0: load part present bit shit with one shot data from the part present sensor
  B3:6/1: ***********************
    Part Width and  Location
    ***********************
    
    Calculates the position of parts on the top belt by measureing the part width by calculating the number of belt movement pulses that occure when the optic is blocked and then devides that in half and add that to the optic location in the part presnet bit shift when the top optic is cleared.
  B9:0/[N7:47]: Remove any part present signals outside of expected location
  B9:0/[N7:50]: Remove any part present signals outside of expected location
  F19:0: Counter inside of a high speed counter interrupt counts the number of Bit Shifts that need to be processed in order to move the logic with the parts on the conveyor.
  F8:14: **************
    Bottom Top Camera Trigger
    *************
    
    Trigger Bottom Top Camera
  N10:4: test if boxing is connected
  B3:11/3: After initial delay allow blow two start functioning
  RUNG000150-000041: transfer tracked part positon from trigger/acquire to the acquire/result
    capture acquire time
    reset process time
  RUNG000150-000039: Grab trigger/acquire position
    Grab acquire time
  RUNG000150-000038: acquire code
  RUNG000150-000035: fail count
  RUNG000150-000032: pass count
  RUNG000150-000025: pass code / Set pass bit in Bit Shift
    captures result position and processing time
    Unlatch pass bit
  RUNG000150-000018: pass, fail and acquire inputs
  RUNG000150-000016: wiped count
  RUNG000150-000014: clear data for time
  RUNG000150-000013: clear data for aquire time expired
  RUNG000150-000012: wipe stored part data if acq time expires
  RUNG000150-000011: trigger count
  L14:5: on when ok to run, rear off turns both off
  L14:2: off when ok to run
  L14:3: off when ok to run
  L14:8: on when ok for run
  L13:165: maximum q i1
  N7:76: removed relieance on trigger signal
  N197:20/0: Passes deformed head blowoff command to TOP PLC where solenoid output is located.
  L13:163: maximum average q
  L13:162: maximum q
  B3:10/1: prevents momentary signals from box present sensor from tripping the logic for box not present
    
    This is in responce to a problem created by the sensor occasionally turning on as if no box was in its path when there is a box present.
  B3:6/2: IF PROCESSING FAULT OCURES AT COUNTER SENSOR; CLEAR THE BELT OF PASSING DATA
  L14:36: ****************  nEEDS fIXING  **********************
  L14:23: ****************  nEEDS fIXING  **********************
  RUNG000010-000018: Remove any part present signals outside of expected location
  RUNG000010-000014: ****
                      Zeros out the non passing part count when one passes
    ****
  T4:26: Check for buffer reset
  T4:27: Check for buffer reset
  RUNG000125-000011: trigger count
  RUNG000125-000012: wipe stored part data if acq time expires
  RUNG000125-000013: clear data for aquire time expired
  RUNG000125-000014: clear data for time
  RUNG000125-000016: wiped count
  RUNG000125-000018: pass, fail and acquire inputs
  RUNG000125-000025: pass code / Set pass bit in Bit Shift
    captures result position and processing time
    Unlatch pass bit
  RUNG000125-000026: Grab trigger/acquire position
    Grab acquire time
  RUNG000125-000027: transfer tracked part positon from trigger/acquire to the acquire/result
    capture acquire time
    reset process time
  RUNG000125-000029: Set pass bit in Bit Shift
    captures result position and processing time
    Unlatch pass bit

REVISION NOTES
  13: updated count reset
  14: added io moduals
  15: multiple steps toward new hmi integration
  21: test

DATA TABLE (non-zero values as saved)
DATA B3
% B3:0 % 0X3020 0X0020 0X2AC1 0XA000 0XAF26 0X0041 0XE9C0 0X56A5 0X2130 0X000C
% B3:10 % 0X2041 0X0846 0X2000 0X0000 0X0000 0X0000 0X0000 0X0000 0X0000 0X0000
DATA T4
% .PRE .ACC %
% T4:0 % 222 109
% T4:1 % 222 106
% T4:2 % 600 0
% T4:3 % 1000 1000
% T4:4 % 3 0
% T4:5 % 666 0
% T4:6 % 10 32766
% T4:7 % 250 0
% T4:8 % 250 0
% T4:9 % 50 33
% T4:10 % 200 200
% T4:11 % 666 0
% T4:12 % 60 61
% T4:13 % 6 0
% T4:14 % 250 0
% T4:15 % 222 110
% T4:16 % 222 108
% T4:17 % 100 1
% T4:18 % 120 0
% T4:19 % 300 0
% T4:20 % 200 0
% T4:21 % 200 0
% T4:22 % 200 0
% T4:23 % 250 0
% T4:24 % 666 0
% T4:25 % 666 0
% T4:26 % 250 0
% T4:27 % 250 0
% T4:28 % 250 0
% T4:29 % 5000 0
% T4:30 % 50 50
% T4:31 % 20 0
% T4:32 % 69 0
DATA C5
% .PRE .ACC %
% C5:0 % 32766 0
DATA R6
% .LEN .POS %
% R6:0 % 2048 0
% R6:1 % 2048 0
% R6:2 % 3 0
% R6:3 % 3 0
% R6:4 % 1250 0
% R6:5 % 1250 0
% R6:6 % 1100 0
% R6:7 % 10 0
% R6:8 % 3 0
% R6:9 % 3 0
% R6:10 % 1440 0
% R6:11 % 1440 0
% R6:12 % 10 0
% R6:13 % 10 0
% R6:14 % 10 0
% R6:15 % 10 0
% R6:16 % 1100 0
% R6:17 % 1440 0
% R6:18 % 1440 0
% R6:19 % 10 0
DATA N7
% N7:0 % 1035 28 1071 27 0 49 49 28 50 0
% N7:10 % 18 62 0 18 1378 250 777 666 11195 102
% N7:20 % 0 73 0 0 0 29 29 1190 333 20
% N7:30 % 46 10 2 222 222 3 1638 222 1165 222
% N7:40 % 2067 2122 40 20 2102 40 81 2027 80 1647
% N7:50 % 1657 400 20 7 0 0 1662 1680 20 7
% N7:60 % 0 0 1051 20 50 2024 2025 2022 2021 20
% N7:70 % 0 21 23 27738 32767 0 122 0 16 0
% N7:80 % 0 6 95 0 0 0 5 500 0 0
% N7:90 % 2011 4 4 12 1 0 0 0 0 1600
% N7:100 % 1003 90 110 100 175 25 0 0 0 0
DATA F8
% F8:0 % 18 206.64 23807 499 0.23807
% F8:5 % 0 0 500 1.9 2
% F8:10 % 1 0.08897486 0 101 63.26563
% F8:15 % 37.73437 4040 2 0 0
% F8:20 % 0 0.02 0 1 0
% F8:25 % 0 932781 0.222 279.6551 848597
% F8:30 % 0 170 0.03 38 852060
% F8:35 % 0 0 0 0 77
% F8:40 % 101 37.73437 0 100 1
% F8:45 % 1 2 0.21455 0 0
% F8:50 % 0 0 1 0 1
% F8:55 % 2000000 -221 0 0 0
% F8:95 % 0 0 0 492 4.92
DATA B12
% B12:0 % 0X0554 0X0000 0X0000 0X0000 0X0000 0X0000 0X0000 0X0000 0X0000 0X0000
DATA L13
% L13:0 % 308402300 308407124 4824 0 1000
% L13:5 % 4794 -1334860360 100 1162124017 1162124017
% L13:10 % 492 1900 0 0 1350415757
% L13:15 % -1227261957 -2147483648 2147483647 2147483647 82058
% L13:20 % 300000000 2072136995 0 -1313930960 2035272617
% L13:25 % 27 0 1042944 0 1000000000
% L13:30 % -1283018343 0 2044398469 13 0
% L13:35 % 0 0 2044398469 17 2035272617
% L13:40 % -1283018330 0 19 20 0
% L13:45 % 60 400 27 0 16
% L13:50 % 0 20 444 20 3
% L13:55 % 0 0 55756418 20983 225
% L13:60 % 0 10576 13 2044398343 12
% L13:65 % 0 20 -3 15571828 501
% L13:70 % 15597849 15597812 37 0 500
% L13:75 % -1 10 337021 -1313930933 337
% L13:80 % 27 -47 9545 0 99
% L13:85 % 6475 2297 31654 -1283017405 -1283017385
% L13:90 % 26616 0 0 1000 0
% L13:95 % 60 0 0 25989 55755519
% L13:100 % 55755518 -1283017376 -1283017358 2 19
% L13:105 % 2044398942 2044398952 15 23 0
% L13:110 % 0 29 27 2044398346 1711915290
% L13:115 % 2044398343 18 9 2044398343 34
% L13:120 % 29 10576 50 100 27
% L13:125 % 164 2044398942 2044398952 20 20
% L13:130 % 34 0 0 20982 0
% L13:135 % 0 1000 20982 12 0
% L13:140 % 0 0 12 0 20
% L13:145 % 0 27738658 35155 35889 37099
% L13:150 % 5 5 5 5 5
% L13:155 % 5 5 24 0 168160
% L13:160 % 3 5 4 395082 53203921
% L13:165 % 3 189116 95 13 0
% L13:170 % 55946610 0 0 0 0
% L13:175 % 0 0 45 32 38
% L13:180 % 176247033 25 99000 52866 644409
% L13:185 % 64 916459 92 627156 63
% L13:190 % 4 5 0 0 0
DATA F14
% F14:0 % 760.1599 200.1099 76 20 15
% F14:5 % 32766 21297.9 0 0 0
DATA N15
% N15:0 % 6 889 2023 1373 1174 134 65 1172 1048 10
% N15:10 % 61 504 0 0 0 0 1172 0 0 0
DATA L16
% L16:0 % 16 60 11 0 20
% L16:5 % 250 5000 5000 182 19
% L16:10 % 1256 18 2045 6599584 98
% L16:15 % 99 0 0 0 0
DATA B17
% B17:50 % 0X0000 0X0010 0X0000 0X0000 0X0000 0X0000 0X0000 0X0000 0X0000 0X0000
% B17:60 % 0XC000 0X0000 0X0000 0X0000 0X0000 0X0000 0X0000 0X0000 0X0000 0X0000
DATA B18
% B18:50 % 0X0000 0X0010 0X0000 0X0000 0X0000 0X0000 0X0000 0X0000 0X0000 0X0000
% B18:60 % 0XC000 0X0000 0X0000 0X0000 0X0000 0X0000 0X0000 0X0000 0X0000 0X0000
DATA L19
% L19:0 % -1283196654 -1283195323 -1283192058 -1283183350 -1283183075
% L19:5 % -1283181890 -1283180182 -1283166844 -1283166239 -1283165297
% L19:10 % -1283162876 -1283160977 -1283160261 -1283156247 -1283154508
% L19:15 % -1283150762 -1283150545 -1283146037 -1283143756 -1283136773
% L19:20 % -1283135954 -1283134621 -1283130537 -1283124229 -1283119415
% L19:25 % -1283107768 -1283082047 -1283065621 -1283039326 -1283018343
% L19:30 % -1283265370 -1283265083 -1283264582 -1283264271 -1283264007
% L19:35 % -1283263666 -1283263164 -1283262909 -1283262401 -1283261556
% L19:40 % -1283261304 -1283260569 -1283258978 -1283258655 -1283257865
% L19:45 % -1283257591 -1283256554 -1283256298 -1283254701 -1283198965
DATA L20
% L20:0 % 2044308597 2044309268 2044310914 2044315303 2044315442
% L20:5 % 2044316039 2044316900 2044323622 2044323927 2044324402
% L20:10 % 2044325621 2044326578 2044326939 2044328961 2044329837
% L20:15 % 2044331725 2044331834 2044334106 2044335255 2044338775
% L20:20 % 2044339188 2044339860 2044341919 2044345098 2044347524
% L20:25 % 2044353393 2044366358 2044374635 2044387893 2044398469
% L20:30 % 2044273963 2044274108 2044274360 2044274517 2044274650
% L20:35 % 2044274822 2044275075 2044275204 2044275460 2044275886
% L20:40 % 2044276013 2044276383 2044277185 2044277348 2044277746
% L20:45 % 2044277884 2044278407 2044278536 2044279341 2044307432
DATA L21
% L21:0 % -1456642640 -1456630632 -1456629536 -1456628403 -1456586572
% L21:5 % -1456585211 -1456583421 -1456441527 -1456321522 -1374440011
% L21:10 % -1374439785 -1374438436 -1374438211 -1374437986 -1313932980
% L21:15 % -1313932756 -1313931410 -1313931185 -1313930960 -1457121541
% L21:20 % -1457121316 -1457121092 -1457120867 -1457120642 -1457120418
% L21:25 % -1457120193 -1457119969 -1457119744 -1457020348 -1457004417
% L21:30 % -1456982493 -1456827692 -1456788552 -1456784332 -1456781708
% L21:35 % -1456774058 -1456754829 -1456733709 -1456715262 -1456702126
% L21:40 % -1456698983 -1456697952 -1456696835 -1456694985 -1456682086
% L21:45 % -1456681059 -1456679928 -1456678581 -1456645862 -1456644127
DATA L22
% L22:0 % 2033873571 2033877809 2033878196 2033878595 2033893352
% L22:5 % 2033893833 2033894464 2033944528 2033986868 2035216335
% L22:10 % 2035216335 2035216335 2035216335 2035216335 2035272617
% L22:15 % 2035272617 2035272617 2035272617 2035272617 2033705715
% L22:20 % 2033705715 2033705715 2033705715 2033705715 2033705715
% L22:25 % 2033705715 2033705715 2033705715 2033740316 2033745935
% L22:30 % 2033753670 2033808284 2033822093 2033823582 2033824508
% L22:35 % 2033827207 2033833991 2033841442 2033847950 2033852584
% L22:40 % 2033853693 2033854057 2033854451 2033855104 2033859654
% L22:45 % 2033860016 2033860415 2033860890 2033872434 2033873046
DATA L23
% L23:0 % -1283164357 -1283161937 -1283160038 -1283159322 -1283155307
% L23:5 % -1283153568 -1283149823 -1283149607 -1283145098 -1283142817
% L23:10 % -1283135834 -1283135015 -1283133682 -1283129598 -1283123291
% L23:15 % -1283118476 -1283106830 -1283081108 -1283064684 -1283038387
% L23:20 % -1283017405 -1283264431 -1283264144 -1283263644 -1283263332
% L23:25 % -1283263069 -1283262727 -1283262226 -1283261970 -1283261462
% L23:30 % -1283260617 -1283260365 -1283259630 -1283258039 -1283257717
% L23:35 % -1283256927 -1283256653 -1283255616 -1283255360 -1283253762
% L23:40 % -1283198026 -1283195716 -1283194384 -1283191120 -1283182412
% L23:45 % -1283182137 -1283180952 -1283179243 -1283165906 -1283165301
DATA L24
% L24:0 % 2044324875 2044326094 2044327051 2044327412 2044329434
% L24:5 % 2044330310 2044332198 2044332307 2044334579 2044335728
% L24:10 % 2044339248 2044339661 2044340333 2044342392 2044345571
% L24:15 % 2044347997 2044353866 2044366831 2044375108 2044388366
% L24:20 % 2044398942 2044274436 2044274581 2044274833 2044274990
% L24:25 % 2044275123 2044275295 2044275548 2044275677 2044275933
% L24:30 % 2044276359 2044276486 2044276856 2044277658 2044277821
% L24:35 % 2044278219 2044278357 2044278880 2044279009 2044279814
% L24:40 % 2044307905 2044309070 2044309741 2044311387 2044315776
% L24:45 % 2044315915 2044316512 2044317373 2044324095 2044324400
DATA L25
% L25:0 % -1283129578 -1283123271 -1283118457 -1283106810 -1283081088
% L25:5 % -1283064664 -1283038367 -1283017385 -1283264412 -1283264124
% L25:10 % -1283263625 -1283263313 -1283263049 -1283262708 -1283262206
% L25:15 % -1283261951 -1283261442 -1283260597 -1283260345 -1283259611
% L25:20 % -1283258020 -1283257697 -1283256907 -1283256633 -1283255596
% L25:25 % -1283255340 -1283253743 -1283198006 -1283195696 -1283194364
% L25:30 % -1283191100 -1283182393 -1283182117 -1283180932 -1283179223
% L25:35 % -1283165886 -1283165280 -1283164338 -1283161917 -1283160019
% L25:40 % -1283159302 -1283155287 -1283153549 -1283149804 -1283149587
% L25:45 % -1283145078 -1283142797 -1283135815 -1283134995 -1283133663
DATA L26
% L26:0 % 2044342402 2044345581 2044348007 2044353876 2044366841
% L26:5 % 2044375118 2044388376 2044398952 2044274446 2044274591
% L26:10 % 2044274843 2044275000 2044275133 2044275305 2044275558
% L26:15 % 2044275687 2044275943 2044276369 2044276496 2044276866
% L26:20 % 2044277668 2044277831 2044278229 2044278367 2044278890
% L26:25 % 2044279019 2044279824 2044307915 2044309080 2044309751
% L26:30 % 2044311397 2044315786 2044315925 2044316522 2044317383
% L26:35 % 2044324105 2044324410 2044324885 2044326104 2044327061
% L26:40 % 2044327422 2044329444 2044330320 2044332208 2044332317
% L26:45 % 2044334589 2044335738 2044339258 2044339671 2044340343
DATA L27
% L27:0 % -1327737903 -1327409080 -1326531174 -1326503371 -1326384218
% L27:5 % -1326211724 -1324866424 -1324806047 -1324711468 -1324467228
% L27:10 % -1324275206 -1324203819 -1323798609 -1323623923 -1323246073
% L27:15 % -1323224310 -1322769920 -1322539862 -1321835876 -1321753516
% L27:20 % -1321619048 -1321207441 -1320571459 -1318912248 -1316319582
% L27:25 % -1314663010 -1312013172 -1309897222 -1334860360 -1334799186
% L27:30 % -1334770055 -1334719350 -1334687802 -1334661282 -1334627384
% L27:35 % -1334576805 -1334551005 -1334499904 -1334413995 -1334389100
% L27:40 % -1334314729 -1334154648 -1334121673 -1334042154 -1334014330
% L27:45 % -1333910000 -1333884673 -1333723515 -1328104535 -1327871659
DATA L42
% L42:0 % -734706020 256 0 0 0
% L42:5 % 45 45 45 0 0
% L42:20 % 0 0 32766 32766 0
% L42:50 % 0 30
DATA L183
% L183:0 % 1427522383 1427522384 1 1000000000 0
% L183:5 % 321 6 283 0 0
DATA N184
% N184:0 % 0 333 0 0 0 0 0 0 0 0
DATA B185
% B185:0 % 0X0200 0X0001 0X0000 0X0000 0X0000 0X0000 0X0000 0X0000 0X0000 0X0000
DATA N186
% N186:0 % 100 0 0 0 0 0 0 0 0 0
DATA L187
% L187:0 % 34 0 497 0 0
% L187:5 % 1063 0 0 0 0
% L187:20 % 0 134217728 0 0 0
DATA F188
% F188:0 % 6 66 11 44 29
DATA B189
% B189:0 % 0X00F0 0X0000 0X0000 0X0000 0X0000 0X0000 0X0000 0X0000 0X0000 0X0000
DATA L190
% L190:0 % 1 5 0 0 0
% L190:30 % 0 2 0 0 0
DATA B191
% B191:0 % 0X0000 0X0001 0X0000 0X0000 0X0000 0X0000 0X0000 0X0000 0X0000 0X0000
DATA L192
% L192:0 % -1444152502 266932201 5055 76 0
% L192:5 % 1000000 39200000 999 999 8
% L192:10 % 0 0 0 -1 -1
% L192:15 % 15800130 -1 -1 13 0
% L192:20 % -1 26000000 -1 -1 -1
% L192:25 % -1 -1 -1 -1 -1
% L192:30 % -1 -1 -1 -1 -1
% L192:35 % -1 -1 -1 -1 -1
% L192:40 % -1 -1 -1 -1 -1
% L192:45 % -1 -1 -1 -1 -1
DATA F193
% F193:0 % nan nan nan nan nan
% F193:5 % nan nan nan nan nan
% F193:10 % nan nan nan nan nan
% F193:15 % nan nan nan nan nan
% F193:20 % nan nan nan nan nan
% F193:25 % nan nan nan nan nan
% F193:30 % nan nan nan nan nan
% F193:35 % nan nan nan nan nan
% F193:40 % nan nan nan nan nan
% F193:45 % nan nan nan nan nan
DATA B196
% B196:0 % 0X0224 0X9FF2 0X0001 0X0000 0X0000 0X0000 0X0000 0X0000 0X0000 0X0000
% B196:30 % 0XE800 0X9BFF 0XEBFF 0XFFDF 0XFFFF 0X0000 0X0000 0X0000 0X0000 0X0000
DATA N197
% N197:0 % 1560 150 500 2500 2500 14417 5555 300 150 0
% N197:10 % 4000 969 4 0 0 0 0 0 0 0
% N197:30 % 15 48 0 0 0 0 0 0 0 0
DATA B198
% B198:0 % 0X0009 0X0000 0X0000 0X0000 0X0000 0X0000 0X0000 0X0000 0X0000 0X0000
DATA L199
% L199:0 % 1 5571998 134 11 3579521
% L199:5 % 0 0 0 5 80526
% L199:10 % 0 224 10256 556 0
% L199:15 % 0 0 0 278717848 518
% L199:20 % 28295 16430853 5001 5001 0
% L199:25 % 0 0 28329 1 3781224
% L199:30 % 21630086 251 3809367 15030467 111
% L199:35 % 555 555 0 0 0
DATA N200
% N200:0 % 2046 1231 985 2047 2045 1594 1241 2045 2045 2045
% N200:10 % 0 0 0 1277 178 2046 1000 2045 2045 1218
% N200:20 % 1555 0 0 0 0 0 0 0 0 0
% N200:30 % 0 0 32767 0 0 0 0 0 0 0
DATA L201
% L201:0 % 20 40 40 -3011735 44
% L201:5 % 96629277 0 0 -3010662 0
% L201:10 % 0 0 0 327 43
% L201:15 % 0 43 0 43 36830
DATA B202
% B202:0 % 0X2241 0X0000 0X0001 0X0000 0X0000 0X0000 0X0000 0X0000 0X0000 0X0000
DATA N203
% N203:0 % 115 115 116 333 334 333 444 0 445 444
% N203:10 % 555 556 555 0 0 0 0 0 0 0
DATA L204
% L204:0 % 333 333 333 1362 124
% L204:5 % 2000 2000 462 222 0
% L204:10 % 0 0 0 1327077052 1327077052
% L204:15 % 1327077052 1327077052 1 0 0
% L204:20 % 0 0 333 0 0
% L204:30 % 333 0 0 0 0
DATA F205
% F205:0 % 655.32 655.32 655.32 655.32 0
